(* PLC project PLC, Beckhoff Automation GmbH TwinCAT PLC Control 3.5.13.21 *)
(* stored: creationDateTime 2024-02-17T22:42:30.6764627, modificationDateTime 2024-02-17T22:42:30.6764627 *)

TYPE LPStatus :
STRUCT
	name: STRING(G.nameStringLength);
	on: BOOL;
END_STRUCT
END_TYPE
